Fanuc KAREL source: compact_preamble.KL

PROGRAM KT00775
%NOLOCKGROUP
VAR
R1:REAL;R2:REAL;OUT:REAL
BEGIN
R1=2.0
R2=3.0
R1=2.0
R2=3.0
OUT=ASIN(R1)
END KT00775
